// TIA Portal V20 export
DATA_BLOCK "DataFromSafety"   // DB127
// stored: Access Published, AssignedProDiagFB Safety.ProDiag, InstanceOfName Safety.typeDataFromSafety, InstanceOfType UDT, Namespace Safety
"Safety.typeDataFromSafety"
   // VAR
   //    devicesSummary { ExternalWritable := 'False'} : "Safety.typeDevicesStatusSummary";
   //    mainOp { ExternalWritable := 'False'} : "Safety.typeMainOpMode";
   //    pHmi { ExternalWritable := 'False'} : "Safety.typePhmi";
   //    scsMode { ExternalWritable := 'False'} : "Safety.typeScsMode";
   //    rcMode1 { ExternalWritable := 'False'} : "Safety.typeRollChangeMode";
   //    rcMode2 { ExternalWritable := 'False'} : "Safety.typeRollChangeMode";
   //    eStopStatus { ExternalWritable := 'False'} : "Safety.typeEstopStatus";
   //    fDoorSwitchStatus { ExternalWritable := 'False'} : "Safety.typeFDoorSwitchStatus";
   //    fDoorCoilStatus { ExternalWritable := 'False'} : "Safety.typeFDoorUnlockOutput";
   //    Zone1SafetyMainOpEnable { ExternalWritable := 'False'} : "Safety.typeSafetyOperationEnable";
   //    Zone1SafetySubOpEnable { S7_SetPoint := 'True'} : "Safety.typeSafetyOperationEnable";
   //    Zone2SafetyOpEnable { ExternalWritable := 'False'} : "Safety.typeSafetyOperationEnable";
   //    Zone3SafetyOpEnable { ExternalWritable := 'False'} : "Safety.typeSafetyOperationEnable";
   //    eStopZone1 { ExternalWritable := 'False'} : "Safety.typeEstopFunction";
   //    eStopZone2 { ExternalWritable := 'False'} : "Safety.typeEstopFunction";
   //    eStopZone3 { ExternalWritable := 'False'} : "Safety.typeEstopFunction";
   //    statusZone1 { ExternalWritable := 'False'} : "Safety.typeSafetyZoneStatus";
   //    statusZone2 { ExternalWritable := 'False'} : "Safety.typeSafetyZoneStatus";
   //    statusZone3 { ExternalWritable := 'False'} : "Safety.typeSafetyZoneStatus";
   //    fDoorDrive : "Safety.typeFDoorFunction";
   //    driveStatus : "Safety.typeSafetyDriveStatus";
   //    SafetySensor { ExternalWritable := 'False'} : "Safety.typeSafetySensor";
   //    FeedbackFault { ExternalWritable := 'False'} : "Safety.typeFeedbackFault";
   //    AllEstopsOK { ExternalWritable := 'False'} : Bool;
   //    allEstopButtonsOK : Bool;
   //    AllEstopsOKfromOther : Bool;
   //    AllFdoorClose { ExternalWritable := 'False'} : Bool;
   //    AllSFDoorOpen { ExternalWritable := 'False'} : Bool;
   //    AnyNoMFDoorOpen { ExternalWritable := 'False'} : Bool;
   //    safetyReleasedAllSafetyZones { ExternalWritable := 'False'} : Bool;
   //    ackRequiredAnySafetyZone { ExternalWritable := 'False'} : Bool;
   //    ackOP_changeRequired { ExternalWritable := 'False'} : Bool;
   //    ackOperatorControlCondition : Bool;
   //    doorBoxAllReset : Bool;
   //    totalSafetyReset { ExternalAccessible := 'False'; ExternalVisible := 'False'; ExternalWritable := 'False'} : Bool;
   //    zone1DoorOpenRequest : Bool;
   //    zone2DoorOpenRequest : Bool;
   //    zone3DoorOpenRequest : Bool;
   //    zone1DriveAckReq : Bool;
   //    zone2DriveAckReq : Bool;
   //    zone3DriveAckReq : Bool;
   //    noSafetyFault : Bool;
   //    ConnectionBoxID { ExternalWritable := 'False'} : Int;
   //    BA60jrPPLeftDoorForcedOpen : Bool;
   //    BA060STOP : Bool;
   //    BA60LightCurtainMuttingRequest : Bool;
   //    BA60LightCurtainDetect : Bool;
   //    BA60RequestForEntry : Bool;
   //    BA60ExternalDoorOpen : Bool;
   //    BA60jrPPLeftDoorNormalOpen : Bool;
   //    PhmiConnectedToBA60 : Bool;
   //    PhmiEnableToBA60 : Bool;
   //    HmiEnableToBA60 : Bool;
   //    BA40CathodeCoverClose : Bool;
   //    BA40AnodeCoverClose : Bool;
   //    BA60Stacker2LightCurtainDetect : Bool;
   //    BA60Stacker2MaintanceDoorOpen : Bool;
   //    SS1TimeExtension : Bool;
   //    EnableServoAck : Bool;
   //    SetupModeFault : Bool;
   //    CathodeCoverSensorFault : Bool;
   //    AnodeCoverSensorFault : Bool;
   //    Door02UnlockPB : Bool;
   //    Door03UnlockPB : Bool;
   //    Door04UnlockPB : Bool;
   //    Door05UnlockPB : Bool;
   //    BA10 { ExternalWritable := 'False'} : "Safety.typeDataFlinkUsed";
   //    BA15 { ExternalWritable := 'False'} : "Safety.typeDataFlinkUsed";
   //    BA40 { ExternalWritable := 'False'} : "Safety.typeDataFlinkUsed";
   //    BA60 { ExternalWritable := 'False'} : "Safety.typeDataFlinkUsed";
   //    cvCoverStatus { ExternalWritable := 'False'} : "Safety.typeCvCoverStatus";
   //    hotWireCutterStatus { ExternalWritable := 'False'} : "Safety.typeHotWireCutter";
   //    fDoorUnwinderTopDoorOpenWarning { ExternalWritable := 'False'} : Bool;
   //    fDoorUnwinderBtmDoorOpenWarning { ExternalWritable := 'False'} : Bool;
   //    PhmiForcedDisconnection : Bool;
   //    CathodeConveyorCoverClosedCheck : Bool;
   //    AnodeConveyorCoverClosedCheck : Bool;
   //    FDoorForcedOpenStatus : "Safety.typeSafetyForcedDoorOpen";
   // END_VAR
BEGIN
END_DATA_BLOCK
